TYPE RobotState :
STRUCT
	joints_position : Joints;
	cartesian_position : Cartesian;
	joints_setpoint : Joints;
	cartesian_setpoint : Cartesian;
END_STRUCT
END_TYPE

(* stored: Version 1.1.0.1, ProductVersion 3.1.4024.10
   DUT RobotState: Id {729d144b-a755-481f-abb3-37ff2995d7bc} *)
